ABB RobotStudio station: Convey_tracking.rsstn

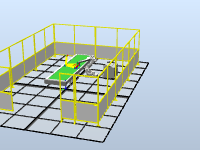
Station Solution16 (saved by RobotStudio 6.8.8307.1040)
Controller System1, task T_ROB1: task frame (RAPID world) sits at (1751.76, 0, 375) mm in the station
Controller System1
  mechanical unit ROB_1: IRB1520ID_4_150__02, 6 joints, base frame (220.19, -534.84, -375) mm, rotated rx 0 ry 0 rz 90 deg
  mechanical unit CNV1: ?, 1 joints, base frame (0, 0, 0) mm
Layout (positions relative to the parent item):
  - IRB1520ID_4_150__02 [mechanism, from Robots\IRB1520ID_4_150_G_02.rslib] at (1971.95, -534.84, 0) mm, rotated rx 0 ry 0 rz 90 deg; joint values [0.323, -0.8091, 1.0617, -0.5438, 0.8515, 0.9505] (rad or m)
  - MyTool [mechanism, from Training Objects\myTool.rslib] at (1862.17, 38.45, 715.53) mm, rotated rx -180 ry 38 rz -110.71 deg
  - Conveyor [conveyor]
    - Convey [part] at (51.76, 0, 375) mm
    - Text_A_1 [part] at (1768.49, 227.97, 415) mm
  - 950_4000_h2 [part, from Equipment\Conveyor 950 4000 h2.rslib]
  - fence [graphiccomponentgroup, from Libraries\fence.rslib] at (-1500, 0, 0) mm
    - Fence_2500_1 [graphiccomponentgroup, from Equipment\Fence_2500.rslib] at (6000, 0, 0) mm
      - Body 1 [part, from Equipment\Fence_2500.rslib]
      - Body 2 [part, from Equipment\Fence_2500.rslib]
    - Fence_2500_2 [graphiccomponentgroup, from Equipment\Fence_2500.rslib] at (6000, -2500, 0) mm
      - Body 1 [part, from Equipment\Fence_2500.rslib]
      - Body 2 [part, from Equipment\Fence_2500.rslib]
    - Fence_2500_3 [graphiccomponentgroup, from Equipment\Fence_2500.rslib] at (6000, 2500, 0) mm, rotated rx 0 ry 0 rz 90 deg
      - Body 1 [part, from Equipment\Fence_2500.rslib]
      - Body 2 [part, from Equipment\Fence_2500.rslib]
    - Fence_2500_4 [graphiccomponentgroup, from Equipment\Fence_2500.rslib] at (6000, -2500, 0) mm, rotated rx 0 ry 0 rz 90 deg
      - Body 1 [part, from Equipment\Fence_2500.rslib]
      - Body 2 [part, from Equipment\Fence_2500.rslib]
    - Fence_2500_5 [graphiccomponentgroup, from Equipment\Fence_2500.rslib] at (3500, 2500, 0) mm, rotated rx 0 ry 0 rz 90 deg
      - Body 1 [part, from Equipment\Fence_2500.rslib]
      - Body 2 [part, from Equipment\Fence_2500.rslib]
    - Fence_2500_6 [graphiccomponentgroup, from Equipment\Fence_2500.rslib] at (3500, -2500, 0) mm, rotated rx 0 ry 0 rz 90 deg
      - Body 1 [part, from Equipment\Fence_2500.rslib]
      - Body 2 [part, from Equipment\Fence_2500.rslib]
    - Fence_2500_7 [graphiccomponentgroup, from Equipment\Fence_2500.rslib] at (1000, -2500, 0) mm, rotated rx 0 ry 0 rz 90 deg
      - Body 1 [part, from Equipment\Fence_2500.rslib]
      - Body 2 [part, from Equipment\Fence_2500.rslib]
    - Fence_2500_8 [graphiccomponentgroup, from Equipment\Fence_2500.rslib] at (1000, 2500, 0) mm, rotated rx 0 ry 0 rz 90 deg
      - Body 1 [part, from Equipment\Fence_2500.rslib]
      - Body 2 [part, from Equipment\Fence_2500.rslib]
    - Fence_Gate [graphiccomponentgroup, from Equipment\Fence_Gate.rslib] at (-1500, 2500, 0) mm, rotated rx 0 ry 0 rz 180 deg
      - Body 1 [part, from Equipment\Fence_Gate.rslib]
      - Body 2 [part, from Equipment\Fence_Gate.rslib]
      - Body 3 [part, from Equipment\Fence_Gate.rslib]
    - Fence_Gate_1 [graphiccomponentgroup, from Equipment\Fence_Gate.rslib] at (-1500, -1040, 0) mm, rotated rx 0 ry 0 rz 180 deg
      - Body 1 [part, from Equipment\Fence_Gate.rslib]
      - Body 2 [part, from Equipment\Fence_Gate.rslib]
      - Body 3 [part, from Equipment\Fence_Gate.rslib]
  - IRC5_Control-Module [part, from Equipment\IRC5_Control-Module.rslib] at (2206.8, -1403.62, 100) mm, rotated rx 90 ry 0 rz 180 deg
Attachment: MyTool is attached to IRB1520ID_4_150__02 / Link6
Conveyor tracking Connection: unit CNV1, TravelOffset=1.7, QueueTrackDistance=0, StartWindowWidth=0.01, SyncSeparation=5E-06, CountsPerMeter=20000
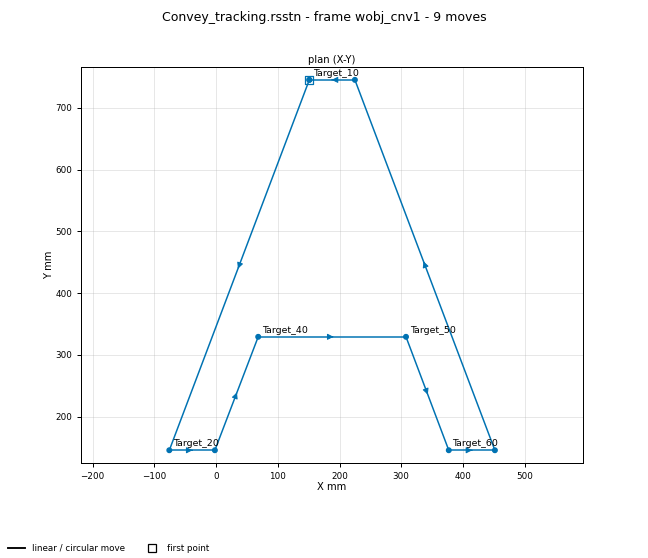
[picture p0: tool path of Convey_tracking.rsstn in frame wobj_cnv1, 9 of 11 moves have a stored position in this frame; points joined in program order, loops and branches not executed]
Targets, tools, work objects and paths stored in the station, written as RAPID:
! task T_ROB1
MODULE CalibData
  PERS tooldata MyTool:=[TRUE,[[31.792631019,0,229.638935148],[0.945518576,0,0.325568154,0]],[1,[0,0,1],[1,0,0,0],0,0,0]];
  TASK PERS wobjdata wobj_cnv1:=[FALSE,FALSE,"CNV1",[[0,0,0],[1,0,0,0]],[[0,0,0],[1,0,0,0]]];
ENDMODULE

! task T_ROB1
MODULE Module1
  CONST robtarget Home:=[[220.185851205,704.339573237,625.64730631],[0.134922335,-0.694115238,0.694115238,0.134922335],[0,-1,0,0],[9E+09,9E+09,9E+09,9E+09,9E+09,0]];
  CONST robtarget Target_10:=[[151.11640625,745.39,140],[0,-0.568504684,0.822680025,0],[0,0,0,0],[9E+09,9E+09,9E+09,9E+09,9E+09,0]];
  CONST robtarget Target_20:=[[-75.7,145.39,140],[0,-0.568504684,0.822680025,0],[0,0,0,0],[9E+09,9E+09,9E+09,9E+09,9E+09,0]];
  CONST robtarget Target_30:=[[-1.901171875,145.39,140],[0,-0.568504684,0.822680025,0],[0,0,0,0],[9E+09,9E+09,9E+09,9E+09,9E+09,0]];
  CONST robtarget Target_40:=[[68.294140625,329.14,140],[0,-0.568504684,0.822680025,0],[0,0,0,0],[9E+09,9E+09,9E+09,9E+09,9E+09,0]];
  CONST robtarget Target_50:=[[307.708203125,329.14,140],[0,-0.568504684,0.822680025,0],[0,0,0,0],[9E+09,9E+09,9E+09,9E+09,9E+09,0]];
  CONST robtarget Target_60:=[[376.9953125,145.39,140],[0,-0.568504684,0.822680025,0],[0,0,0,0],[9E+09,9E+09,9E+09,9E+09,9E+09,0]];
  CONST robtarget Target_70:=[[451.70234375,145.39,140],[0,-0.568504684,0.822680025,0],[0,0,0,0],[9E+09,9E+09,9E+09,9E+09,9E+09,0]];
  CONST robtarget Target_80:=[[224.915234375,745.39,140],[0,-0.568504684,0.822680025,0],[0,0,0,0],[9E+09,9E+09,9E+09,9E+09,9E+09,0]];
  CONST robtarget Target_90:=[[151.11640625,745.39,140],[0,-0.568504684,0.822680025,0],[0,0,0,0],[9E+09,9E+09,9E+09,9E+09,9E+09,0]];
  PROC Path_10()
    MoveL Home,v1000,z100,MyTool\WObj:=wobj0;
    ActUnit CNV1;
    WaitWObj wobj_cnv1;
    MoveL Target_10,v5000,fine,MyTool\WObj:=wobj_cnv1;
    MoveL Target_20,v5000,fine,MyTool\WObj:=wobj_cnv1;
    MoveL Target_30,v5000,fine,MyTool\WObj:=wobj_cnv1;
    MoveL Target_40,v5000,fine,MyTool\WObj:=wobj_cnv1;
    MoveL Target_50,v5000,fine,MyTool\WObj:=wobj_cnv1;
    MoveL Target_60,v5000,fine,MyTool\WObj:=wobj_cnv1;
    MoveL Target_70,v5000,fine,MyTool\WObj:=wobj_cnv1;
    MoveL Target_80,v5000,fine,MyTool\WObj:=wobj_cnv1;
    MoveL Target_90,v5000,fine,MyTool\WObj:=wobj_cnv1;
    MoveL Home,v1000,z100,MyTool\WObj:=wobj0;
    DropWObj wobj_cnv1;
  ENDPROC
ENDMODULE

